D10852	WORD	Память для хранения названий рецептов. Задание 54. Символы 9-10
D10853	WORD	Память для хранения названий рецептов. Задание 54. Символы 11-12
D10854	WORD	Память для хранения названий рецептов. Задание 54. Символы 13-14
D10855	WORD	Память для хранения названий рецептов. Задание 54. Символы 15-16
D10856	WORD	Память для хранения названий рецептов. Задание 54. Символы 17-18
D10857	WORD	Память для хранения названий рецептов. Задание 54. Символы 19-20
D10858	WORD	Память для хранения названий рецептов. Задание 54. Символы 21-22
D10859	WORD	Память для хранения названий рецептов. Задание 54. Символы 23-24
D10860	WORD	Память для хранения названий рецептов. Задание 54. Символы 25-26
D10861	WORD	Память для хранения названий рецептов. Задание 54. Символы 27-28
D10862	WORD	Память для хранения названий рецептов. Задание 54. Символы 29-30
D10863	WORD	Память для хранения названий рецептов. Задание 54. Символы 31-32
D10864	WORD	Память для хранения названий рецептов. Задание 55. Символы 1-2
D10865	WORD	Память для хранения названий рецептов. Задание 55. Символы 3-4
D10866	WORD	Память для хранения названий рецептов. Задание 55. Символы 5-6
D10867	WORD	Память для хранения названий рецептов. Задание 55. Символы 7-8
D10868	WORD	Память для хранения названий рецептов. Задание 55. Символы 9-10
D10869	WORD	Память для хранения названий рецептов. Задание 55. Символы 11-12
D10870	WORD	Память для хранения названий рецептов. Задание 55. Символы 13-14
D10871	WORD	Память для хранения названий рецептов. Задание 55. Символы 15-16
D10872	WORD	Память для хранения названий рецептов. Задание 55. Символы 17-18
D10873	WORD	Память для хранения названий рецептов. Задание 55. Символы 19-20
D10874	WORD	Память для хранения названий рецептов. Задание 55. Символы 21-22
D10875	WORD	Память для хранения названий рецептов. Задание 55. Символы 23-24
D10876	WORD	Память для хранения названий рецептов. Задание 55. Символы 25-26
D10877	WORD	Память для хранения названий рецептов. Задание 55. Символы 27-28
D10878	WORD	Память для хранения названий рецептов. Задание 55. Символы 29-30
D10879	WORD	Память для хранения названий рецептов. Задание 55. Символы 31-32
D10880	WORD	Память для хранения названий рецептов. Задание 56. Символы 1-2
D10881	WORD	Память для хранения названий рецептов. Задание 56. Символы 3-4
D10882	WORD	Память для хранения названий рецептов. Задание 56. Символы 5-6
D10883	WORD	Память для хранения названий рецептов. Задание 56. Символы 7-8
D10884	WORD	Память для хранения названий рецептов. Задание 56. Символы 9-10
D10885	WORD	Память для хранения названий рецептов. Задание 56. Символы 11-12
D10886	WORD	Память для хранения названий рецептов. Задание 56. Символы 13-14
D10887	WORD	Память для хранения названий рецептов. Задание 56. Символы 15-16
D10888	WORD	Память для хранения названий рецептов. Задание 56. Символы 17-18
D10889	WORD	Память для хранения названий рецептов. Задание 56. Символы 19-20
D10890	WORD	Память для хранения названий рецептов. Задание 56. Символы 21-22
D10891	WORD	Память для хранения названий рецептов. Задание 56. Символы 23-24
D10892	WORD	Память для хранения названий рецептов. Задание 56. Символы 25-26
D10893	WORD	Память для хранения названий рецептов. Задание 56. Символы 27-28
D10894	WORD	Память для хранения названий рецептов. Задание 56. Символы 29-30
D10895	WORD	Память для хранения названий рецептов. Задание 56. Символы 31-32
D10896	WORD	Память для хранения названий рецептов. Задание 57. Символы 1-2
D10897	WORD	Память для хранения названий рецептов. Задание 57. Символы 3-4
D10898	WORD	Память для хранения названий рецептов. Задание 57. Символы 5-6
D10899	WORD	Память для хранения названий рецептов. Задание 57. Символы 7-8
D10900	WORD	Память для хранения названий рецептов. Задание 57. Символы 9-10
D10901	WORD	Память для хранения названий рецептов. Задание 57. Символы 11-12
D10902	WORD	Память для хранения названий рецептов. Задание 57. Символы 13-14
D10903	WORD	Память для хранения названий рецептов. Задание 57. Символы 15-16
D10904	WORD	Память для хранения названий рецептов. Задание 57. Символы 17-18
D10905	WORD	Память для хранения названий рецептов. Задание 57. Символы 19-20
D10906	WORD	Память для хранения названий рецептов. Задание 57. Символы 21-22
D10907	WORD	Память для хранения названий рецептов. Задание 57. Символы 23-24
D10908	WORD	Память для хранения названий рецептов. Задание 57. Символы 25-26
D10909	WORD	Память для хранения названий рецептов. Задание 57. Символы 27-28
D10910	WORD	Память для хранения названий рецептов. Задание 57. Символы 29-30
D10911	WORD	Память для хранения названий рецептов. Задание 57. Символы 31-32
D10912	WORD	Память для хранения названий рецептов. Задание 58. Символы 1-2
D10913	WORD	Память для хранения названий рецептов. Задание 58. Символы 3-4
D10914	WORD	Память для хранения названий рецептов. Задание 58. Символы 5-6
D10915	WORD	Память для хранения названий рецептов. Задание 58. Символы 7-8
D10916	WORD	Память для хранения названий рецептов. Задание 58. Символы 9-10
D10917	WORD	Память для хранения названий рецептов. Задание 58. Символы 11-12
D10918	WORD	Память для хранения названий рецептов. Задание 58. Символы 13-14
D10919	WORD	Память для хранения названий рецептов. Задание 58. Символы 15-16
D10920	WORD	Память для хранения названий рецептов. Задание 58. Символы 17-18
D10921	WORD	Память для хранения названий рецептов. Задание 58. Символы 19-20
D10922	WORD	Память для хранения названий рецептов. Задание 58. Символы 21-22
D10923	WORD	Память для хранения названий рецептов. Задание 58. Символы 23-24
D10924	WORD	Память для хранения названий рецептов. Задание 58. Символы 25-26
D10925	WORD	Память для хранения названий рецептов. Задание 58. Символы 27-28
D10926	WORD	Память для хранения названий рецептов. Задание 58. Символы 29-30
D10927	WORD	Память для хранения названий рецептов. Задание 58. Символы 31-32
D10928	WORD	Память для хранения названий рецептов. Задание 59. Символы 1-2
D10929	WORD	Память для хранения названий рецептов. Задание 59. Символы 3-4
D10930	WORD	Память для хранения названий рецептов. Задание 59. Символы 5-6
D10931	WORD	Память для хранения названий рецептов. Задание 59. Символы 7-8
D10932	WORD	Память для хранения названий рецептов. Задание 59. Символы 9-10
D10933	WORD	Память для хранения названий рецептов. Задание 59. Символы 11-12
D10934	WORD	Память для хранения названий рецептов. Задание 59. Символы 13-14
D10935	WORD	Память для хранения названий рецептов. Задание 59. Символы 15-16
D10936	WORD	Память для хранения названий рецептов. Задание 59. Символы 17-18
D10937	WORD	Память для хранения названий рецептов. Задание 59. Символы 19-20
D10938	WORD	Память для хранения названий рецептов. Задание 59. Символы 21-22
D10939	WORD	Память для хранения названий рецептов. Задание 59. Символы 23-24
D10940	WORD	Память для хранения названий рецептов. Задание 59. Символы 25-26
D10941	WORD	Память для хранения названий рецептов. Задание 59. Символы 27-28
D10942	WORD	Память для хранения названий рецептов. Задание 59. Символы 29-30
D10943	WORD	Память для хранения названий рецептов. Задание 59. Символы 31-32
D10944	WORD	Память для хранения названий рецептов. Задание 60. Символы 1-2
D10945	WORD	Память для хранения названий рецептов. Задание 60. Символы 3-4
D10946	WORD	Память для хранения названий рецептов. Задание 60. Символы 5-6
D10947	WORD	Память для хранения названий рецептов. Задание 60. Символы 7-8
D10948	WORD	Память для хранения названий рецептов. Задание 60. Символы 9-10
D10949	WORD	Память для хранения названий рецептов. Задание 60. Символы 11-12
D10950	WORD	Память для хранения названий рецептов. Задание 60. Символы 13-14
D10951	WORD	Память для хранения названий рецептов. Задание 60. Символы 15-16
D10952	WORD	Память для хранения названий рецептов. Задание 60. Символы 17-18
D10953	WORD	Память для хранения названий рецептов. Задание 60. Символы 19-20
D10954	WORD	Память для хранения названий рецептов. Задание 60. Символы 21-22
D10955	WORD	Память для хранения названий рецептов. Задание 60. Символы 23-24
D10956	WORD	Память для хранения названий рецептов. Задание 60. Символы 25-26
D10957	WORD	Память для хранения названий рецептов. Задание 60. Символы 27-28
D10958	WORD	Память для хранения названий рецептов. Задание 60. Символы 29-30
D10959	WORD	Память для хранения названий рецептов. Задание 60. Символы 31-32
D11001	WORD	Память для хранения названий рецептов. Пластина 1. Символы 3-4
D11002	WORD	Память для хранения названий рецептов. Пластина 1. Символы 5-6
D11003	WORD	Память для хранения названий рецептов. Пластина 1. Символы 7-8
D11004	WORD	Память для хранения названий рецептов. Пластина 1. Символы 9-10
D11005	WORD	Память для хранения названий рецептов. Пластина 1. Символы 11-12
D11006	WORD	Память для хранения названий рецептов. Пластина 1. Символы 13-14
D11007	WORD	Память для хранения названий рецептов. Пластина 1. Символы 15-16
D11008	WORD	Память для хранения названий рецептов. Пластина 1. Символы 17-18
D11009	WORD	Память для хранения названий рецептов. Пластина 1. Символы 19-20
D11010	WORD	Память для хранения названий рецептов. Пластина 1. Символы 21-22
D11011	WORD	Память для хранения названий рецептов. Пластина 1. Символы 23-24
D11012	WORD	Память для хранения названий рецептов. Пластина 1. Символы 25-26
D11013	WORD	Память для хранения названий рецептов. Пластина 1. Символы 27-28
D11014	WORD	Память для хранения названий рецептов. Пластина 1. Символы 29-30
D11015	WORD	Память для хранения названий рецептов. Пластина 1. Символы 31-32
D11016	WORD	Память для хранения названий рецептов. Пластина 2. Символы 1-2
D11017	WORD	Память для хранения названий рецептов. Пластина 2. Символы 3-4
D11018	WORD	Память для хранения названий рецептов. Пластина 2. Символы 5-6
D11019	WORD	Память для хранения названий рецептов. Пластина 2. Символы 7-8
D11020	WORD	Память для хранения названий рецептов. Пластина 2. Символы 9-10
D11021	WORD	Память для хранения названий рецептов. Пластина 2. Символы 11-12
D11022	WORD	Память для хранения названий рецептов. Пластина 2. Символы 13-14
D11023	WORD	Память для хранения названий рецептов. Пластина 2. Символы 15-16
D11024	WORD	Память для хранения названий рецептов. Пластина 2. Символы 17-18
D11025	WORD	Память для хранения названий рецептов. Пластина 2. Символы 19-20
D11026	WORD	Память для хранения названий рецептов. Пластина 2. Символы 21-22
D11027	WORD	Память для хранения названий рецептов. Пластина 2. Символы 23-24
D11028	WORD	Память для хранения названий рецептов. Пластина 2. Символы 25-26
D11029	WORD	Память для хранения названий рецептов. Пластина 2. Символы 27-28
D11030	WORD	Память для хранения названий рецептов. Пластина 2. Символы 29-30
D11031	WORD	Память для хранения названий рецептов. Пластина 2. Символы 31-32
D11032	WORD	Память для хранения названий рецептов. Пластина 3. Символы 1-2
D11033	WORD	Память для хранения названий рецептов. Пластина 3. Символы 3-4
D11034	WORD	Память для хранения названий рецептов. Пластина 3. Символы 5-6
D11035	WORD	Память для хранения названий рецептов. Пластина 3. Символы 7-8
D11036	WORD	Память для хранения названий рецептов. Пластина 3. Символы 9-10
D11037	WORD	Память для хранения названий рецептов. Пластина 3. Символы 11-12
D11038	WORD	Память для хранения названий рецептов. Пластина 3. Символы 13-14
D11039	WORD	Память для хранения названий рецептов. Пластина 3. Символы 15-16
D11040	WORD	Память для хранения названий рецептов. Пластина 3. Символы 17-18
D11041	WORD	Память для хранения названий рецептов. Пластина 3. Символы 19-20
D11042	WORD	Память для хранения названий рецептов. Пластина 3. Символы 21-22
D11043	WORD	Память для хранения названий рецептов. Пластина 3. Символы 23-24
D11044	WORD	Память для хранения названий рецептов. Пластина 3. Символы 25-26
D11045	WORD	Память для хранения названий рецептов. Пластина 3. Символы 27-28
D11046	WORD	Память для хранения названий рецептов. Пластина 3. Символы 29-30
D11047	WORD	Память для хранения названий рецептов. Пластина 3. Символы 31-32
D11048	WORD	Память для хранения названий рецептов. Пластина 4. Символы 1-2
D11049	WORD	Память для хранения названий рецептов. Пластина 4. Символы 3-4
D11050	WORD	Память для хранения названий рецептов. Пластина 4. Символы 5-6
D11051	WORD	Память для хранения названий рецептов. Пластина 4. Символы 7-8
D11052	WORD	Память для хранения названий рецептов. Пластина 4. Символы 9-10
D11053	WORD	Память для хранения названий рецептов. Пластина 4. Символы 11-12
D11054	WORD	Память для хранения названий рецептов. Пластина 4. Символы 13-14
D11055	WORD	Память для хранения названий рецептов. Пластина 4. Символы 15-16
D11056	WORD	Память для хранения названий рецептов. Пластина 4. Символы 17-18
D11057	WORD	Память для хранения названий рецептов. Пластина 4. Символы 19-20
D11058	WORD	Память для хранения названий рецептов. Пластина 4. Символы 21-22
D11059	WORD	Память для хранения названий рецептов. Пластина 4. Символы 23-24
D11060	WORD	Память для хранения названий рецептов. Пластина 4. Символы 25-26
D11061	WORD	Память для хранения названий рецептов. Пластина 4. Символы 27-28
D11062	WORD	Память для хранения названий рецептов. Пластина 4. Символы 29-30
D11063	WORD	Память для хранения названий рецептов. Пластина 4. Символы 31-32
D11064	WORD	Память для хранения названий рецептов. Пластина 5. Символы 1-2
D11065	WORD	Память для хранения названий рецептов. Пластина 5. Символы 3-4
D11066	WORD	Память для хранения названий рецептов. Пластина 5. Символы 5-6
D11067	WORD	Память для хранения названий рецептов. Пластина 5. Символы 7-8
D11068	WORD	Память для хранения названий рецептов. Пластина 5. Символы 9-10
D11069	WORD	Память для хранения названий рецептов. Пластина 5. Символы 11-12
D11070	WORD	Память для хранения названий рецептов. Пластина 5. Символы 13-14
D11071	WORD	Память для хранения названий рецептов. Пластина 5. Символы 15-16
D11072	WORD	Память для хранения названий рецептов. Пластина 5. Символы 17-18
D11073	WORD	Память для хранения названий рецептов. Пластина 5. Символы 19-20
D11074	WORD	Память для хранения названий рецептов. Пластина 5. Символы 21-22
D11075	WORD	Память для хранения названий рецептов. Пластина 5. Символы 23-24
D11076	WORD	Память для хранения названий рецептов. Пластина 5. Символы 25-26
D11077	WORD	Память для хранения названий рецептов. Пластина 5. Символы 27-28
D11078	WORD	Память для хранения названий рецептов. Пластина 5. Символы 29-30
D11079	WORD	Память для хранения названий рецептов. Пластина 5. Символы 31-32
D11080	WORD	Память для хранения названий рецептов. Пластина 6. Символы 1-2
D11081	WORD	Память для хранения названий рецептов. Пластина 6. Символы 3-4
D11082	WORD	Память для хранения названий рецептов. Пластина 6. Символы 5-6
D11083	WORD	Память для хранения названий рецептов. Пластина 6. Символы 7-8
D11084	WORD	Память для хранения названий рецептов. Пластина 6. Символы 9-10
D11085	WORD	Память для хранения названий рецептов. Пластина 6. Символы 11-12
D11086	WORD	Память для хранения названий рецептов. Пластина 6. Символы 13-14
D11087	WORD	Память для хранения названий рецептов. Пластина 6. Символы 15-16
D11088	WORD	Память для хранения названий рецептов. Пластина 6. Символы 17-18
D11089	WORD	Память для хранения названий рецептов. Пластина 6. Символы 19-20
D11090	WORD	Память для хранения названий рецептов. Пластина 6. Символы 21-22
D11091	WORD	Память для хранения названий рецептов. Пластина 6. Символы 23-24
D11092	WORD	Память для хранения названий рецептов. Пластина 6. Символы 25-26
D11093	WORD	Память для хранения названий рецептов. Пластина 6. Символы 27-28
D11094	WORD	Память для хранения названий рецептов. Пластина 6. Символы 29-30
D11095	WORD	Память для хранения названий рецептов. Пластина 6. Символы 31-32
D11096	WORD	Память для хранения названий рецептов. Пластина 7. Символы 1-2
D11097	WORD	Память для хранения названий рецептов. Пластина 7. Символы 3-4
D11098	WORD	Память для хранения названий рецептов. Пластина 7. Символы 5-6
D11099	WORD	Память для хранения названий рецептов. Пластина 7. Символы 7-8
D11100	WORD	Память для хранения названий рецептов. Пластина 7. Символы 9-10
D11101	WORD	Память для хранения названий рецептов. Пластина 7. Символы 11-12
D11102	WORD	Память для хранения названий рецептов. Пластина 7. Символы 13-14
D11103	WORD	Память для хранения названий рецептов. Пластина 7. Символы 15-16
D11104	WORD	Память для хранения названий рецептов. Пластина 7. Символы 17-18
D11105	WORD	Память для хранения названий рецептов. Пластина 7. Символы 19-20
D11106	WORD	Память для хранения названий рецептов. Пластина 7. Символы 21-22
D11107	WORD	Память для хранения названий рецептов. Пластина 7. Символы 23-24
D11108	WORD	Память для хранения названий рецептов. Пластина 7. Символы 25-26
D11109	WORD	Память для хранения названий рецептов. Пластина 7. Символы 27-28
D11110	WORD	Память для хранения названий рецептов. Пластина 7. Символы 29-30
D11111	WORD	Память для хранения названий рецептов. Пластина 7. Символы 31-32
D11112	WORD	Память для хранения названий рецептов. Пластина 8. Символы 1-2
D11113	WORD	Память для хранения названий рецептов. Пластина 8. Символы 3-4
D11114	WORD	Память для хранения названий рецептов. Пластина 8. Символы 5-6
D11115	WORD	Память для хранения названий рецептов. Пластина 8. Символы 7-8
D11116	WORD	Память для хранения названий рецептов. Пластина 8. Символы 9-10
D11117	WORD	Память для хранения названий рецептов. Пластина 8. Символы 11-12
D11118	WORD	Память для хранения названий рецептов. Пластина 8. Символы 13-14
D11119	WORD	Память для хранения названий рецептов. Пластина 8. Символы 15-16
D11120	WORD	Память для хранения названий рецептов. Пластина 8. Символы 17-18
D11121	WORD	Память для хранения названий рецептов. Пластина 8. Символы 19-20
D11122	WORD	Память для хранения названий рецептов. Пластина 8. Символы 21-22
D11123	WORD	Память для хранения названий рецептов. Пластина 8. Символы 23-24
D11124	WORD	Память для хранения названий рецептов. Пластина 8. Символы 25-26
D11125	WORD	Память для хранения названий рецептов. Пластина 8. Символы 27-28
D11126	WORD	Память для хранения названий рецептов. Пластина 8. Символы 29-30
D11127	WORD	Память для хранения названий рецептов. Пластина 8. Символы 31-32
D11128	WORD	Память для хранения названий рецептов. Пластина 9. Символы 1-2
D11129	WORD	Память для хранения названий рецептов. Пластина 9. Символы 3-4
D11130	WORD	Память для хранения названий рецептов. Пластина 9. Символы 5-6
D11131	WORD	Память для хранения названий рецептов. Пластина 9. Символы 7-8
D11132	WORD	Память для хранения названий рецептов. Пластина 9. Символы 9-10
D11133	WORD	Память для хранения названий рецептов. Пластина 9. Символы 11-12
D11134	WORD	Память для хранения названий рецептов. Пластина 9. Символы 13-14
D11135	WORD	Память для хранения названий рецептов. Пластина 9. Символы 15-16
D11136	WORD	Память для хранения названий рецептов. Пластина 9. Символы 17-18
D11137	WORD	Память для хранения названий рецептов. Пластина 9. Символы 19-20
D11138	WORD	Память для хранения названий рецептов. Пластина 9. Символы 21-22
D11139	WORD	Память для хранения названий рецептов. Пластина 9. Символы 23-24
D11140	WORD	Память для хранения названий рецептов. Пластина 9. Символы 25-26
D11141	WORD	Память для хранения названий рецептов. Пластина 9. Символы 27-28
D11142	WORD	Память для хранения названий рецептов. Пластина 9. Символы 29-30
D11143	WORD	Память для хранения названий рецептов. Пластина 9. Символы 31-32
D11144	WORD	Память для хранения названий рецептов. Пластина 10. Символы 1-2
D11145	WORD	Память для хранения названий рецептов. Пластина 10. Символы 3-4
D11146	WORD	Память для хранения названий рецептов. Пластина 10. Символы 5-6
D11147	WORD	Память для хранения названий рецептов. Пластина 10. Символы 7-8
D11148	WORD	Память для хранения названий рецептов. Пластина 10. Символы 9-10
D11149	WORD	Память для хранения названий рецептов. Пластина 10. Символы 11-12
D11150	WORD	Память для хранения названий рецептов. Пластина 10. Символы 13-14
D11151	WORD	Память для хранения названий рецептов. Пластина 10. Символы 15-16
D11152	WORD	Память для хранения названий рецептов. Пластина 10. Символы 17-18
D11153	WORD	Память для хранения названий рецептов. Пластина 10. Символы 19-20
D11154	WORD	Память для хранения названий рецептов. Пластина 10. Символы 21-22
D11155	WORD	Память для хранения названий рецептов. Пластина 10. Символы 23-24
D11156	WORD	Память для хранения названий рецептов. Пластина 10. Символы 25-26
D11157	WORD	Память для хранения названий рецептов. Пластина 10. Символы 27-28
D11158	WORD	Память для хранения названий рецептов. Пластина 10. Символы 29-30
D11159	WORD	Память для хранения названий рецептов. Пластина 10. Символы 31-32
D11160	WORD	Память для хранения названий рецептов. Пластина 11. Символы 1-2
D11161	WORD	Память для хранения названий рецептов. Пластина 11. Символы 3-4
D11162	WORD	Память для хранения названий рецептов. Пластина 11. Символы 5-6
D11163	WORD	Память для хранения названий рецептов. Пластина 11. Символы 7-8
D11164	WORD	Память для хранения названий рецептов. Пластина 11. Символы 9-10
D11165	WORD	Память для хранения названий рецептов. Пластина 11. Символы 11-12
D11166	WORD	Память для хранения названий рецептов. Пластина 11. Символы 13-14
D11167	WORD	Память для хранения названий рецептов. Пластина 11. Символы 15-16
D11168	WORD	Память для хранения названий рецептов. Пластина 11. Символы 17-18
D11169	WORD	Память для хранения названий рецептов. Пластина 11. Символы 19-20
D11170	WORD	Память для хранения названий рецептов. Пластина 11. Символы 21-22
D11171	WORD	Память для хранения названий рецептов. Пластина 11. Символы 23-24
D11172	WORD	Память для хранения названий рецептов. Пластина 11. Символы 25-26
D11173	WORD	Память для хранения названий рецептов. Пластина 11. Символы 27-28
D11174	WORD	Память для хранения названий рецептов. Пластина 11. Символы 29-30
D11175	WORD	Память для хранения названий рецептов. Пластина 11. Символы 31-32
D11176	WORD	Память для хранения названий рецептов. Пластина 12. Символы 1-2
D11177	WORD	Память для хранения названий рецептов. Пластина 12. Символы 3-4
D11178	WORD	Память для хранения названий рецептов. Пластина 12. Символы 5-6
D11179	WORD	Память для хранения названий рецептов. Пластина 12. Символы 7-8
D11180	WORD	Память для хранения названий рецептов. Пластина 12. Символы 9-10
D11181	WORD	Память для хранения названий рецептов. Пластина 12. Символы 11-12
D11182	WORD	Память для хранения названий рецептов. Пластина 12. Символы 13-14
D11183	WORD	Память для хранения названий рецептов. Пластина 12. Символы 15-16
D11184	WORD	Память для хранения названий рецептов. Пластина 12. Символы 17-18
D11185	WORD	Память для хранения названий рецептов. Пластина 12. Символы 19-20
D11186	WORD	Память для хранения названий рецептов. Пластина 12. Символы 21-22
D11187	WORD	Память для хранения названий рецептов. Пластина 12. Символы 23-24
D11188	WORD	Память для хранения названий рецептов. Пластина 12. Символы 25-26
D11189	WORD	Память для хранения названий рецептов. Пластина 12. Символы 27-28
D11190	WORD	Память для хранения названий рецептов. Пластина 12. Символы 29-30
D11191	WORD	Память для хранения названий рецептов. Пластина 12. Символы 31-32
D11192	WORD	Память для хранения названий рецептов. Пластина 13. Символы 1-2
D11193	WORD	Память для хранения названий рецептов. Пластина 13. Символы 3-4
D11194	WORD	Память для хранения названий рецептов. Пластина 13. Символы 5-6
D11195	WORD	Память для хранения названий рецептов. Пластина 13. Символы 7-8
D11196	WORD	Память для хранения названий рецептов. Пластина 13. Символы 9-10
D11197	WORD	Память для хранения названий рецептов. Пластина 13. Символы 11-12
D11198	WORD	Память для хранения названий рецептов. Пластина 13. Символы 13-14
D11199	WORD	Память для хранения названий рецептов. Пластина 13. Символы 15-16
D11200	WORD	Память для хранения названий рецептов. Пластина 13. Символы 17-18
D11201	WORD	Память для хранения названий рецептов. Пластина 13. Символы 19-20
D11202	WORD	Память для хранения названий рецептов. Пластина 13. Символы 21-22
D11203	WORD	Память для хранения названий рецептов. Пластина 13. Символы 23-24
D11204	WORD	Память для хранения названий рецептов. Пластина 13. Символы 25-26
D11205	WORD	Память для хранения названий рецептов. Пластина 13. Символы 27-28
D11206	WORD	Память для хранения названий рецептов. Пластина 13. Символы 29-30
D11207	WORD	Память для хранения названий рецептов. Пластина 13. Символы 31-32
D11208	WORD	Память для хранения названий рецептов. Пластина 14. Символы 1-2
D11209	WORD	Память для хранения названий рецептов. Пластина 14. Символы 3-4
D11210	WORD	Память для хранения названий рецептов. Пластина 14. Символы 5-6
D11211	WORD	Память для хранения названий рецептов. Пластина 14. Символы 7-8
D11212	WORD	Память для хранения названий рецептов. Пластина 14. Символы 9-10
D11213	WORD	Память для хранения названий рецептов. Пластина 14. Символы 11-12
D11214	WORD	Память для хранения названий рецептов. Пластина 14. Символы 13-14
D11215	WORD	Память для хранения названий рецептов. Пластина 14. Символы 15-16
D11216	WORD	Память для хранения названий рецептов. Пластина 14. Символы 17-18
D11217	WORD	Память для хранения названий рецептов. Пластина 14. Символы 19-20
D11218	WORD	Память для хранения названий рецептов. Пластина 14. Символы 21-22
D11219	WORD	Память для хранения названий рецептов. Пластина 14. Символы 23-24
D11220	WORD	Память для хранения названий рецептов. Пластина 14. Символы 25-26
D11221	WORD	Память для хранения названий рецептов. Пластина 14. Символы 27-28
D11222	WORD	Память для хранения названий рецептов. Пластина 14. Символы 29-30
D11223	WORD	Память для хранения названий рецептов. Пластина 14. Символы 31-32
D11224	WORD	Память для хранения названий рецептов. Пластина 15. Символы 1-2
D11225	WORD	Память для хранения названий рецептов. Пластина 15. Символы 3-4
D11226	WORD	Память для хранения названий рецептов. Пластина 15. Символы 5-6
D11227	WORD	Память для хранения названий рецептов. Пластина 15. Символы 7-8
D11228	WORD	Память для хранения названий рецептов. Пластина 15. Символы 9-10
D11229	WORD	Память для хранения названий рецептов. Пластина 15. Символы 11-12
D11230	WORD	Память для хранения названий рецептов. Пластина 15. Символы 13-14
D11231	WORD	Память для хранения названий рецептов. Пластина 15. Символы 15-16
D11232	WORD	Память для хранения названий рецептов. Пластина 15. Символы 17-18
D11233	WORD	Память для хранения названий рецептов. Пластина 15. Символы 19-20
D11234	WORD	Память для хранения названий рецептов. Пластина 15. Символы 21-22
D11235	WORD	Память для хранения названий рецептов. Пластина 15. Символы 23-24
D11236	WORD	Память для хранения названий рецептов. Пластина 15. Символы 25-26
D11237	WORD	Память для хранения названий рецептов. Пластина 15. Символы 27-28
D11238	WORD	Память для хранения названий рецептов. Пластина 15. Символы 29-30
D11239	WORD	Память для хранения названий рецептов. Пластина 15. Символы 31-32
D11240	WORD	Память для хранения названий рецептов. Пластина 16. Символы 1-2
D11241	WORD	Память для хранения названий рецептов. Пластина 16. Символы 3-4
D11242	WORD	Память для хранения названий рецептов. Пластина 16. Символы 5-6
D11243	WORD	Память для хранения названий рецептов. Пластина 16. Символы 7-8
D11244	WORD	Память для хранения названий рецептов. Пластина 16. Символы 9-10
D11245	WORD	Память для хранения названий рецептов. Пластина 16. Символы 11-12
D11246	WORD	Память для хранения названий рецептов. Пластина 16. Символы 13-14
D11247	WORD	Память для хранения названий рецептов. Пластина 16. Символы 15-16
D11248	WORD	Память для хранения названий рецептов. Пластина 16. Символы 17-18
D11249	WORD	Память для хранения названий рецептов. Пластина 16. Символы 19-20
D11250	WORD	Память для хранения названий рецептов. Пластина 16. Символы 21-22
D11251	WORD	Память для хранения названий рецептов. Пластина 16. Символы 23-24
D11252	WORD	Память для хранения названий рецептов. Пластина 16. Символы 25-26
D11253	WORD	Память для хранения названий рецептов. Пластина 16. Символы 27-28
D11254	WORD	Память для хранения названий рецептов. Пластина 16. Символы 29-30
D11255	WORD	Память для хранения названий рецептов. Пластина 16. Символы 31-32
D11256	WORD	Память для хранения названий рецептов. Пластина 17. Символы 1-2
D11257	WORD	Память для хранения названий рецептов. Пластина 17. Символы 3-4
D11258	WORD	Память для хранения названий рецептов. Пластина 17. Символы 5-6
D11259	WORD	Память для хранения названий рецептов. Пластина 17. Символы 7-8
D11260	WORD	Память для хранения названий рецептов. Пластина 17. Символы 9-10
D11261	WORD	Память для хранения названий рецептов. Пластина 17. Символы 11-12
D11262	WORD	Память для хранения названий рецептов. Пластина 17. Символы 13-14
D11263	WORD	Память для хранения названий рецептов. Пластина 17. Символы 15-16
D11264	WORD	Память для хранения названий рецептов. Пластина 17. Символы 17-18
D11265	WORD	Память для хранения названий рецептов. Пластина 17. Символы 19-20
D11266	WORD	Память для хранения названий рецептов. Пластина 17. Символы 21-22
D11267	WORD	Память для хранения названий рецептов. Пластина 17. Символы 23-24
D11268	WORD	Память для хранения названий рецептов. Пластина 17. Символы 25-26
D11269	WORD	Память для хранения названий рецептов. Пластина 17. Символы 27-28
D11270	WORD	Память для хранения названий рецептов. Пластина 17. Символы 29-30
D11271	WORD	Память для хранения названий рецептов. Пластина 17. Символы 31-32
D11272	WORD	Память для хранения названий рецептов. Пластина 18. Символы 1-2
D11273	WORD	Память для хранения названий рецептов. Пластина 18. Символы 3-4
D11274	WORD	Память для хранения названий рецептов. Пластина 18. Символы 5-6
D11275	WORD	Память для хранения названий рецептов. Пластина 18. Символы 7-8
D11276	WORD	Память для хранения названий рецептов. Пластина 18. Символы 9-10
D11277	WORD	Память для хранения названий рецептов. Пластина 18. Символы 11-12
D11278	WORD	Память для хранения названий рецептов. Пластина 18. Символы 13-14
D11279	WORD	Память для хранения названий рецептов. Пластина 18. Символы 15-16
D11280	WORD	Память для хранения названий рецептов. Пластина 18. Символы 17-18
D11281	WORD	Память для хранения названий рецептов. Пластина 18. Символы 19-20
D11282	WORD	Память для хранения названий рецептов. Пластина 18. Символы 21-22
D11283	WORD	Память для хранения названий рецептов. Пластина 18. Символы 23-24
D11284	WORD	Память для хранения названий рецептов. Пластина 18. Символы 25-26
D11285	WORD	Память для хранения названий рецептов. Пластина 18. Символы 27-28
D11286	WORD	Память для хранения названий рецептов. Пластина 18. Символы 29-30
D11287	WORD	Память для хранения названий рецептов. Пластина 18. Символы 31-32
D11288	WORD	Память для хранения названий рецептов. Пластина 19. Символы 1-2
D11289	WORD	Память для хранения названий рецептов. Пластина 19. Символы 3-4
D11290	WORD	Память для хранения названий рецептов. Пластина 19. Символы 5-6
D11291	WORD	Память для хранения названий рецептов. Пластина 19. Символы 7-8
D11292	WORD	Память для хранения названий рецептов. Пластина 19. Символы 9-10
D11293	WORD	Память для хранения названий рецептов. Пластина 19. Символы 11-12
D11294	WORD	Память для хранения названий рецептов. Пластина 19. Символы 13-14
D11295	WORD	Память для хранения названий рецептов. Пластина 19. Символы 15-16
D11296	WORD	Память для хранения названий рецептов. Пластина 19. Символы 17-18
D11297	WORD	Память для хранения названий рецептов. Пластина 19. Символы 19-20
D11298	WORD	Память для хранения названий рецептов. Пластина 19. Символы 21-22
D11299	WORD	Память для хранения названий рецептов. Пластина 19. Символы 23-24
D11300	WORD	Память для хранения названий рецептов. Пластина 19. Символы 25-26
D11301	WORD	Память для хранения названий рецептов. Пластина 19. Символы 27-28
D11302	WORD	Память для хранения названий рецептов. Пластина 19. Символы 29-30
D11303	WORD	Память для хранения названий рецептов. Пластина 19. Символы 31-32
D11304	WORD	Память для хранения названий рецептов. Пластина 20. Символы 1-2
D11305	WORD	Память для хранения названий рецептов. Пластина 20. Символы 3-4
D11306	WORD	Память для хранения названий рецептов. Пластина 20. Символы 5-6
D11307	WORD	Память для хранения названий рецептов. Пластина 20. Символы 7-8
D11308	WORD	Память для хранения названий рецептов. Пластина 20. Символы 9-10
D11309	WORD	Память для хранения названий рецептов. Пластина 20. Символы 11-12
D11310	WORD	Память для хранения названий рецептов. Пластина 20. Символы 13-14
D11311	WORD	Память для хранения названий рецептов. Пластина 20. Символы 15-16
D11312	WORD	Память для хранения названий рецептов. Пластина 20. Символы 17-18
D11313	WORD	Память для хранения названий рецептов. Пластина 20. Символы 19-20
D11314	WORD	Память для хранения названий рецептов. Пластина 20. Символы 21-22
D11315	WORD	Память для хранения названий рецептов. Пластина 20. Символы 23-24
D11316	WORD	Память для хранения названий рецептов. Пластина 20. Символы 25-26
D11317	WORD	Память для хранения названий рецептов. Пластина 20. Символы 27-28
D11318	WORD	Память для хранения названий рецептов. Пластина 20. Символы 29-30
D11319	WORD	Память для хранения названий рецептов. Пластина 20. Символы 31-32
D11320	WORD	Память для хранения названий рецептов. Пластина 21. Символы 1-2
D11321	WORD	Память для хранения названий рецептов. Пластина 21. Символы 3-4
D11322	WORD	Память для хранения названий рецептов. Пластина 21. Символы 5-6
D11323	WORD	Память для хранения названий рецептов. Пластина 21. Символы 7-8
D11324	WORD	Память для хранения названий рецептов. Пластина 21. Символы 9-10
D11325	WORD	Память для хранения названий рецептов. Пластина 21. Символы 11-12
D11326	WORD	Память для хранения названий рецептов. Пластина 21. Символы 13-14
D11327	WORD	Память для хранения названий рецептов. Пластина 21. Символы 15-16
D11328	WORD	Память для хранения названий рецептов. Пластина 21. Символы 17-18
D11329	WORD	Память для хранения названий рецептов. Пластина 21. Символы 19-20
D11330	WORD	Память для хранения названий рецептов. Пластина 21. Символы 21-22
D11331	WORD	Память для хранения названий рецептов. Пластина 21. Символы 23-24
D11332	WORD	Память для хранения названий рецептов. Пластина 21. Символы 25-26
D11333	WORD	Память для хранения названий рецептов. Пластина 21. Символы 27-28
D11334	WORD	Память для хранения названий рецептов. Пластина 21. Символы 29-30
D11335	WORD	Память для хранения названий рецептов. Пластина 21. Символы 31-32
D11336	WORD	Память для хранения названий рецептов. Пластина 22. Символы 1-2
D11337	WORD	Память для хранения названий рецептов. Пластина 22. Символы 3-4
D11338	WORD	Память для хранения названий рецептов. Пластина 22. Символы 5-6
D11339	WORD	Память для хранения названий рецептов. Пластина 22. Символы 7-8
D11340	WORD	Память для хранения названий рецептов. Пластина 22. Символы 9-10
D11341	WORD	Память для хранения названий рецептов. Пластина 22. Символы 11-12
D11342	WORD	Память для хранения названий рецептов. Пластина 22. Символы 13-14
D11343	WORD	Память для хранения названий рецептов. Пластина 22. Символы 15-16
D11344	WORD	Память для хранения названий рецептов. Пластина 22. Символы 17-18
D11345	WORD	Память для хранения названий рецептов. Пластина 22. Символы 19-20
D11346	WORD	Память для хранения названий рецептов. Пластина 22. Символы 21-22
D11347	WORD	Память для хранения названий рецептов. Пластина 22. Символы 23-24
D11348	WORD	Память для хранения названий рецептов. Пластина 22. Символы 25-26
D11349	WORD	Память для хранения названий рецептов. Пластина 22. Символы 27-28
D11350	WORD	Память для хранения названий рецептов. Пластина 22. Символы 29-30
D11351	WORD	Память для хранения названий рецептов. Пластина 22. Символы 31-32
D11352	WORD	Память для хранения названий рецептов. Пластина 23. Символы 1-2
D11353	WORD	Память для хранения названий рецептов. Пластина 23. Символы 3-4
D11354	WORD	Память для хранения названий рецептов. Пластина 23. Символы 5-6
D11355	WORD	Память для хранения названий рецептов. Пластина 23. Символы 7-8
D11356	WORD	Память для хранения названий рецептов. Пластина 23. Символы 9-10
D11357	WORD	Память для хранения названий рецептов. Пластина 23. Символы 11-12
D11358	WORD	Память для хранения названий рецептов. Пластина 23. Символы 13-14
D11359	WORD	Память для хранения названий рецептов. Пластина 23. Символы 15-16
D11360	WORD	Память для хранения названий рецептов. Пластина 23. Символы 17-18
D11361	WORD	Память для хранения названий рецептов. Пластина 23. Символы 19-20
D11362	WORD	Память для хранения названий рецептов. Пластина 23. Символы 21-22
D11363	WORD	Память для хранения названий рецептов. Пластина 23. Символы 23-24
D11364	WORD	Память для хранения названий рецептов. Пластина 23. Символы 25-26
D11365	WORD	Память для хранения названий рецептов. Пластина 23. Символы 27-28
D11366	WORD	Память для хранения названий рецептов. Пластина 23. Символы 29-30
D11367	WORD	Память для хранения названий рецептов. Пластина 23. Символы 31-32
D11368	WORD	Память для хранения названий рецептов. Пластина 24. Символы 1-2
D11369	WORD	Память для хранения названий рецептов. Пластина 24. Символы 3-4
D11370	WORD	Память для хранения названий рецептов. Пластина 24. Символы 5-6
D11371	WORD	Память для хранения названий рецептов. Пластина 24. Символы 7-8
D11372	WORD	Память для хранения названий рецептов. Пластина 24. Символы 9-10
D11373	WORD	Память для хранения названий рецептов. Пластина 24. Символы 11-12
D11374	WORD	Память для хранения названий рецептов. Пластина 24. Символы 13-14
D11375	WORD	Память для хранения названий рецептов. Пластина 24. Символы 15-16
D11376	WORD	Память для хранения названий рецептов. Пластина 24. Символы 17-18
D11377	WORD	Память для хранения названий рецептов. Пластина 24. Символы 19-20
D11378	WORD	Память для хранения названий рецептов. Пластина 24. Символы 21-22
D11379	WORD	Память для хранения названий рецептов. Пластина 24. Символы 23-24
D11380	WORD	Память для хранения названий рецептов. Пластина 24. Символы 25-26
D11381	WORD	Память для хранения названий рецептов. Пластина 24. Символы 27-28
D11382	WORD	Память для хранения названий рецептов. Пластина 24. Символы 29-30
D11383	WORD	Память для хранения названий рецептов. Пластина 24. Символы 31-32
D11384	WORD	Память для хранения названий рецептов. Пластина 25. Символы 1-2
D11385	WORD	Память для хранения названий рецептов. Пластина 25. Символы 3-4
D11386	WORD	Память для хранения названий рецептов. Пластина 25. Символы 5-6
D11387	WORD	Память для хранения названий рецептов. Пластина 25. Символы 7-8
D11388	WORD	Память для хранения названий рецептов. Пластина 25. Символы 9-10
D11389	WORD	Память для хранения названий рецептов. Пластина 25. Символы 11-12
D11390	WORD	Память для хранения названий рецептов. Пластина 25. Символы 13-14
D11391	WORD	Память для хранения названий рецептов. Пластина 25. Символы 15-16
D11392	WORD	Память для хранения названий рецептов. Пластина 25. Символы 17-18
D11393	WORD	Память для хранения названий рецептов. Пластина 25. Символы 19-20
D11394	WORD	Память для хранения названий рецептов. Пластина 25. Символы 21-22
D11395	WORD	Память для хранения названий рецептов. Пластина 25. Символы 23-24
D11396	WORD	Память для хранения названий рецептов. Пластина 25. Символы 25-26
D11397	WORD	Память для хранения названий рецептов. Пластина 25. Символы 27-28
D11398	WORD	Память для хранения названий рецептов. Пластина 25. Символы 29-30
D11399	WORD	Память для хранения названий рецептов. Пластина 25. Символы 31-32
D11400	WORD	Память для хранения названий рецептов. Пластина 26. Символы 1-2
D11401	WORD	Память для хранения названий рецептов. Пластина 26. Символы 3-4
D11402	WORD	Память для хранения названий рецептов. Пластина 26. Символы 5-6
D11403	WORD	Память для хранения названий рецептов. Пластина 26. Символы 7-8
D11404	WORD	Память для хранения названий рецептов. Пластина 26. Символы 9-10
D11405	WORD	Память для хранения названий рецептов. Пластина 26. Символы 11-12
D11406	WORD	Память для хранения названий рецептов. Пластина 26. Символы 13-14
D11407	WORD	Память для хранения названий рецептов. Пластина 26. Символы 15-16
D11408	WORD	Память для хранения названий рецептов. Пластина 26. Символы 17-18
D11409	WORD	Память для хранения названий рецептов. Пластина 26. Символы 19-20
D11410	WORD	Память для хранения названий рецептов. Пластина 26. Символы 21-22
D11411	WORD	Память для хранения названий рецептов. Пластина 26. Символы 23-24
D11412	WORD	Память для хранения названий рецептов. Пластина 26. Символы 25-26
D11413	WORD	Память для хранения названий рецептов. Пластина 26. Символы 27-28
D11414	WORD	Память для хранения названий рецептов. Пластина 26. Символы 29-30
D11415	WORD	Память для хранения названий рецептов. Пластина 26. Символы 31-32
D11416	WORD	Память для хранения названий рецептов. Пластина 27. Символы 1-2
D11417	WORD	Память для хранения названий рецептов. Пластина 27. Символы 3-4
D11418	WORD	Память для хранения названий рецептов. Пластина 27. Символы 5-6
D11419	WORD	Память для хранения названий рецептов. Пластина 27. Символы 7-8
D11420	WORD	Память для хранения названий рецептов. Пластина 27. Символы 9-10
D11421	WORD	Память для хранения названий рецептов. Пластина 27. Символы 11-12
D11422	WORD	Память для хранения названий рецептов. Пластина 27. Символы 13-14
D11423	WORD	Память для хранения названий рецептов. Пластина 27. Символы 15-16
D11424	WORD	Память для хранения названий рецептов. Пластина 27. Символы 17-18
D11425	WORD	Память для хранения названий рецептов. Пластина 27. Символы 19-20
D11426	WORD	Память для хранения названий рецептов. Пластина 27. Символы 21-22
D11427	WORD	Память для хранения названий рецептов. Пластина 27. Символы 23-24
D11428	WORD	Память для хранения названий рецептов. Пластина 27. Символы 25-26
D11429	WORD	Память для хранения названий рецептов. Пластина 27. Символы 27-28
D11430	WORD	Память для хранения названий рецептов. Пластина 27. Символы 29-30
D11431	WORD	Память для хранения названий рецептов. Пластина 27. Символы 31-32
D11432	WORD	Память для хранения названий рецептов. Пластина 28. Символы 1-2
D11433	WORD	Память для хранения названий рецептов. Пластина 28. Символы 3-4
D11434	WORD	Память для хранения названий рецептов. Пластина 28. Символы 5-6
D11435	WORD	Память для хранения названий рецептов. Пластина 28. Символы 7-8
D11436	WORD	Память для хранения названий рецептов. Пластина 28. Символы 9-10
D11437	WORD	Память для хранения названий рецептов. Пластина 28. Символы 11-12
D11438	WORD	Память для хранения названий рецептов. Пластина 28. Символы 13-14
D11439	WORD	Память для хранения названий рецептов. Пластина 28. Символы 15-16
D11440	WORD	Память для хранения названий рецептов. Пластина 28. Символы 17-18
D11441	WORD	Память для хранения названий рецептов. Пластина 28. Символы 19-20
D11442	WORD	Память для хранения названий рецептов. Пластина 28. Символы 21-22
D11443	WORD	Память для хранения названий рецептов. Пластина 28. Символы 23-24
D11444	WORD	Память для хранения названий рецептов. Пластина 28. Символы 25-26
D11445	WORD	Память для хранения названий рецептов. Пластина 28. Символы 27-28
D11446	WORD	Память для хранения названий рецептов. Пластина 28. Символы 29-30
D11447	WORD	Память для хранения названий рецептов. Пластина 28. Символы 31-32
D11448	WORD	Память для хранения названий рецептов. Пластина 29. Символы 1-2
D11449	WORD	Память для хранения названий рецептов. Пластина 29. Символы 3-4
D11450	WORD	Память для хранения названий рецептов. Пластина 29. Символы 5-6
D11451	WORD	Память для хранения названий рецептов. Пластина 29. Символы 7-8
D11452	WORD	Память для хранения названий рецептов. Пластина 29. Символы 9-10
D11453	WORD	Память для хранения названий рецептов. Пластина 29. Символы 11-12
D11454	WORD	Память для хранения названий рецептов. Пластина 29. Символы 13-14
D11455	WORD	Память для хранения названий рецептов. Пластина 29. Символы 15-16
D11456	WORD	Память для хранения названий рецептов. Пластина 29. Символы 17-18
D11457	WORD	Память для хранения названий рецептов. Пластина 29. Символы 19-20
D11458	WORD	Память для хранения названий рецептов. Пластина 29. Символы 21-22
D11459	WORD	Память для хранения названий рецептов. Пластина 29. Символы 23-24
D11460	WORD	Память для хранения названий рецептов. Пластина 29. Символы 25-26
D11461	WORD	Память для хранения названий рецептов. Пластина 29. Символы 27-28
D11462	WORD	Память для хранения названий рецептов. Пластина 29. Символы 29-30
D11463	WORD	Память для хранения названий рецептов. Пластина 29. Символы 31-32
D11464	WORD	Память для хранения названий рецептов. Пластина 30. Символы 1-2
D11465	WORD	Память для хранения названий рецептов. Пластина 30. Символы 3-4
D11466	WORD	Память для хранения названий рецептов. Пластина 30. Символы 5-6
D11467	WORD	Память для хранения названий рецептов. Пластина 30. Символы 7-8
D11468	WORD	Память для хранения названий рецептов. Пластина 30. Символы 9-10
D11469	WORD	Память для хранения названий рецептов. Пластина 30. Символы 11-12
D11470	WORD	Память для хранения названий рецептов. Пластина 30. Символы 13-14
D11471	WORD	Память для хранения названий рецептов. Пластина 30. Символы 15-16
D11472	WORD	Память для хранения названий рецептов. Пластина 30. Символы 17-18
D11473	WORD	Память для хранения названий рецептов. Пластина 30. Символы 19-20
D11474	WORD	Память для хранения названий рецептов. Пластина 30. Символы 21-22
D11475	WORD	Память для хранения названий рецептов. Пластина 30. Символы 23-24
D11476	WORD	Память для хранения названий рецептов. Пластина 30. Символы 25-26
D11477	WORD	Память для хранения названий рецептов. Пластина 30. Символы 27-28
D11478	WORD	Память для хранения названий рецептов. Пластина 30. Символы 29-30
D11479	WORD	Память для хранения названий рецептов. Пластина 30. Символы 31-32
D11480	WORD	Память для хранения названий рецептов. Пластина 31. Символы 1-2
D11481	WORD	Память для хранения названий рецептов. Пластина 31. Символы 3-4
D11482	WORD	Память для хранения названий рецептов. Пластина 31. Символы 5-6
D11483	WORD	Память для хранения названий рецептов. Пластина 31. Символы 7-8
D11484	WORD	Память для хранения названий рецептов. Пластина 31. Символы 9-10
D11485	WORD	Память для хранения названий рецептов. Пластина 31. Символы 11-12
D11486	WORD	Память для хранения названий рецептов. Пластина 31. Символы 13-14
D11487	WORD	Память для хранения названий рецептов. Пластина 31. Символы 15-16
D11488	WORD	Память для хранения названий рецептов. Пластина 31. Символы 17-18
D11489	WORD	Память для хранения названий рецептов. Пластина 31. Символы 19-20
D11490	WORD	Память для хранения названий рецептов. Пластина 31. Символы 21-22
D11491	WORD	Память для хранения названий рецептов. Пластина 31. Символы 23-24
D11492	WORD	Память для хранения названий рецептов. Пластина 31. Символы 25-26
D11493	WORD	Память для хранения названий рецептов. Пластина 31. Символы 27-28
D11494	WORD	Память для хранения названий рецептов. Пластина 31. Символы 29-30
D11495	WORD	Память для хранения названий рецептов. Пластина 31. Символы 31-32
D11496	WORD	Память для хранения названий рецептов. Пластина 32. Символы 1-2
D11497	WORD	Память для хранения названий рецептов. Пластина 32. Символы 3-4
D11498	WORD	Память для хранения названий рецептов. Пластина 32. Символы 5-6
D11499	WORD	Память для хранения названий рецептов. Пластина 32. Символы 7-8
D11500	WORD	Память для хранения названий рецептов. Пластина 32. Символы 9-10
D11501	WORD	Память для хранения названий рецептов. Пластина 32. Символы 11-12
D11502	WORD	Память для хранения названий рецептов. Пластина 32. Символы 13-14
D11503	WORD	Память для хранения названий рецептов. Пластина 32. Символы 15-16
D11504	WORD	Память для хранения названий рецептов. Пластина 32. Символы 17-18
D11505	WORD	Память для хранения названий рецептов. Пластина 32. Символы 19-20
D11506	WORD	Память для хранения названий рецептов. Пластина 32. Символы 21-22
D11507	WORD	Память для хранения названий рецептов. Пластина 32. Символы 23-24
D11508	WORD	Память для хранения названий рецептов. Пластина 32. Символы 25-26
D11509	WORD	Память для хранения названий рецептов. Пластина 32. Символы 27-28
D11510	WORD	Память для хранения названий рецептов. Пластина 32. Символы 29-30
D11511	WORD	Память для хранения названий рецептов. Пластина 32. Символы 31-32
D00171	WORD	Предыдущая выбранная пластина 
T0012	BIT/WORD	100MS Время на смену номера блока и номера рецепта
T0015	BIT/WORD	100MS Таймер сброса команды загрузки данных
T0016	BIT/WORD	100MS Таймер сброса команды сохранения данных
T0017	BIT/WORD	100MS Время на смену номера блока и номера рецепта
T0018	BIT/WORD	100MS Время на смену номера блока и номера рецепта
D00168	WORD	Смещение номера ред. пластины на 100
D00173	WORD	Номер редактируемой пластины -101
D00301	WORD	Диаметр заготовки
D00303	WORD	Диаметр детали
D00305	WORD	Диаметр полуфабриката
D00315	WORD	Обдув патрона перед установкой
D00316	WORD	Обдув патрона после захвата детали
D00317	WORD	Каким захватом берём заготовку
D00318	WORD	В какой патрон ставим заготовку
D00319	WORD	Каким захватом забираем деталь
D00401	WORD	Количество ячеек в нечётных рядах
D00402	WORD	Количество ячеек в чётных рядах
T0019	BIT/WORD	100MS Время на смену номера блока и номера рецепта
D00180	WORD	Последняя загруженная пластина
D00176	WORD	MULNULL
D00177	WORD	MULNULL
D00178	WORD	MULNULL
D00322	WORD	Что сначала: открытие захвата или закрытие патрона 